// SYNTAX TEST "Step7 AWL.sublime-syntax"

// ==================================================
//  common
//  Performance: 3.0ms
// ==================================================

///////////////////////////////////////////////////////////////////////////////
// datatypes                                                                 //
///////////////////////////////////////////////////////////////////////////////

  TYPE "UDT_TypeName"
//^^^^^^^^^^^^^^^^^^^^ meta.block.udt.header
//^^^^ keyword.other.udt.begin
//     ^ punctuation.definition.string.begin
//     ^^^^^^^^^^^^^^ string.quoted.double
//                  ^ punctuation.definition.string.end
   { S7_language illegal := '7(1) Deutsch (Deutschland)  19.01.2014  10:33:55' }
// ^^^^^^^^^^^^^^^^^^^^^^^^^^^^^^^^^^^^^^^^^^^^^^^^^^^^^^^^^^^^^^^^^^^^^^^^^^^^^ meta.block.udt.header
// ^ meta.mapping - meta.mapping.key - meta.mapping.value
//  ^^^^^^^^^^^^^^^^^^^^^ meta.mapping.key - meta.mapping.value
//                       ^^ meta.mapping - meta.mapping.key - meta.mapping.value
//                         ^^^^^^^^^^^^^^^^^^^^^^^^^^^^^^^^^^^^^^^^^^^^^^^^^^^^ meta.mapping.value
//                                                                             ^ meta.mapping - meta.mapping.key - meta.mapping.value
// ^ punctuation.section.mapping.begin
//   ^^^^^^^^^^^ variable.annotation
//               ^^^^^^^ invalid.illegal.separator-expected
//                       ^^ punctuation.separator.key-value
//                                                                             ^ punctuation.section.mapping.end
   NON_RETAIN
// ^^^^^^^^^^ invalid.illegal
   READ_ONLY
// ^^^^^^^^^ invalid.illegal
   VERSION : 1.0
// ^^^^^^^^^^^^^ meta.block.udt.header
// ^^^^^^^^^ meta.mapping.key - meta.mapping.value
//          ^^^^ meta.mapping.value
// ^^^^^^^ entity.other.attribute-name
//         ^ punctuation.separator.key-value
//           ^ constant.numeric.float.version.major
//            ^ punctuation.separator.decimal.version
//             ^ constant.numeric.float.version.minor
   AUTHOR : name
// ^^^^^^^^^^^^^ meta.block.udt.header
// ^^^^^^^^ meta.mapping.key - meta.mapping.value
//         ^^^^^ meta.mapping.value
// ^^^^^^ entity.other.attribute-name
//        ^ punctuation.separator.key-value
//          ^^^^ string.unquoted
   FAMILY : name
// ^^^^^^^^^^^^^ meta.block.udt.header
// ^^^^^^^^ meta.mapping.key - meta.mapping.value
//         ^^^^^ meta.mapping.value
// ^^^^^^ entity.other.attribute-name
//        ^ punctuation.separator.key-value
//          ^^^^ string.unquoted
   NAME : name
// ^^^^^^^^^^^ meta.block.udt.header
// ^^^^^^ meta.mapping.key - meta.mapping.value
//       ^^^^^ meta.mapping.value
// ^^^^ entity.other.attribute-name
//      ^ punctuation.separator.key-value
//        ^^^^ string.unquoted
   ILLEGAL : unknown
// ^^^^^^^^^^^^^^^^^ meta.block.udt.header
// ^^^^^^^ invalid.illegal
//         ^ invalid.illegal
//           ^^^^^^^ invalid.illegal
  STRUCT
//^^^^^^^ meta.block.udt.header meta.struct
//^^^^^^ storage.type.struct.begin
     ID  : INT := 20 ;  //integer
// ^^^^^^^^^^^^^^^^^^^^^^^^^^^^^^^ meta.block.udt.header.s7.awl meta.struct.s7.awl
//   ^^^^^ meta.definition.variable - meta.definition.variable.storage
//        ^^^^^ meta.definition.variable.storage
//             ^^ meta.definition.variable - meta.definition.variable.storage - meta.definition.variable.value
//               ^^^^ meta.definition.variable.value
//   ^^ variable.other
//       ^ punctuation.separator.key-value
//         ^^^ storage.type.integer
//             ^^ keyword.operator.assignment
//                ^^ constant.numeric.integer
//                   ^ punctuation.terminator.statement
//                    ^^ - invalid
//                      ^^^^^^^^^ comment.line.double-slash
//                               ^ - invalid
     PTR : POINTER := P#0.0;
// ^^^^^^^^^^^^^^^^^^^^^^^^^^ meta.block.udt.header.s7.awl meta.struct.s7.awl
//   ^^^^^ meta.definition.variable.s7.awl
//        ^^^^^^^^^ meta.definition.variable.storage.s7.awl
//                 ^^ meta.definition.variable.s7.awl
//                   ^^^^^^ meta.definition.variable.value.s7.awl
//   ^^^ variable.other.s7.awl
//       ^ punctuation.separator.key-value.s7.awl
//         ^^^^^^^ storage.type.pointer.s7.awl
//                 ^^ keyword.operator.assignment.s7.awl
//                    ^^^^^ constant.language.pointer.s7.awl
     TMR : TIMER := T0;
// ^^^^^^^^^^^^^^^^^^^^^ meta.block.udt.header.s7.awl meta.struct.s7.awl
//   ^^^^^ meta.definition.variable.s7.awl
//        ^^^^^^^ meta.definition.variable.storage.s7.awl
//               ^^ meta.definition.variable.s7.awl
//                 ^^^ meta.definition.variable.value.s7.awl
//   ^^^ variable.other.s7.awl
//       ^ punctuation.separator.key-value.s7.awl
//         ^^^^^ storage.type.timer.s7.awl
//               ^^ keyword.operator.assignment.s7.awl
//                  ^^ variable.language.timer.s7.awl
  END_STRUCT ;
//^^^^^^^^^^^^^ meta.block.udt.header
//^^^^^^^^^^ meta.struct storage.type.struct.end
//           ^ punctuation.terminator.statement
  BEGIN
//^^^^^^ meta.block.udt.header
//^^^^^ invalid.illegal
  END_TYPE
//^^^^^^^^ meta.block.udt.header
//^^^^^^^^ keyword.other.udt.end

///////////////////////////////////////////////////////////////////////////////
// datablocks                                                                //
///////////////////////////////////////////////////////////////////////////////

  DATA_BLOCK "name" // comment
// ^^^^^^^^^^^^^^^^^^^^^^^^^^^ meta.block.db.header
// ^^^^^^^^^ keyword.other.db.begin
//           ^ punctuation.definition.string.begin
//           ^^^^^^ string.quoted.double
//            ^^^^ entity.name.block
//                  ^^ punctuation.definition.comment.begin
//                  ^^^^^^^^^^ comment.line.double-slash
   TITLE =the datablock description
// ^^^^^^^^^^^^^^^^^^^^^^^^^^^^^^^^ meta.block.db.header
// ^^^^^^^ meta.mapping.key - meta.mapping.value
//        ^^^^^^^^^^^^^^^^^^^^^^^^ meta.mapping.value - meta.mapping.key
// ^^^^^ entity.other.attribute-name.title
//       ^ punctuation.separator.key-value.title
//        ^^^^^^^^^^^^^^^^^^^^^^^^^ entity.name.section.s7.awl
   { S7_language illegal := '7(1) Deutsch (Deutschland)  19.01.2014  10:33:55' }
// ^^^^^^^^^^^^^^^^^^^^^^^^^^^^^^^^^^^^^^^^^^^^^^^^^^^^^^^^^^^^^^^^^^^^^^^^^^^^^ meta.block.db.header
// ^ meta.mapping - meta.mapping.key - meta.mapping.value
//  ^^^^^^^^^^^^^^^^^^^^^ meta.mapping.key - meta.mapping.value
//                       ^^ meta.mapping - meta.mapping.key - meta.mapping.value
//                         ^^^^^^^^^^^^^^^^^^^^^^^^^^^^^^^^^^^^^^^^^^^^^^^^^^^^ meta.mapping.value
//                                                                             ^ meta.mapping - meta.mapping.key - meta.mapping.value
// ^ punctuation.section.mapping.begin
//   ^^^^^^^^^^^ variable.annotation
//               ^^^^^^^ invalid.illegal.separator-expected
//                       ^^ punctuation.separator.key-value
//                                                                             ^ punctuation.section.mapping.end
   NON_RETAIN
// ^^^^^^^^^^ entity.other.attribute-name
   READ_ONLY
// ^^^^^^^^^ entity.other.attribute-name
   VERSION : 1.0
// ^^^^^^^^^^^^^ meta.block.db.header
// ^^^^^^^^^ meta.mapping.key - meta.mapping.value
//          ^^^^ meta.mapping.value
// ^^^^^^^ entity.other.attribute-name
//         ^ punctuation.separator.key-value
//           ^ constant.numeric.float.version.major
//            ^ punctuation.separator.decimal.version
//             ^ constant.numeric.float.version.minor
   AUTHOR : name
// ^^^^^^^^^^^^^ meta.block.db.header
// ^^^^^^^^ meta.mapping.key - meta.mapping.value
//         ^^^^^ meta.mapping.value
// ^^^^^^ entity.other.attribute-name
//        ^ punctuation.separator.key-value
//          ^^^^ string.unquoted
   FAMILY : name
// ^^^^^^^^^^^^^ meta.block.db.header
// ^^^^^^^^ meta.mapping.key - meta.mapping.value
//         ^^^^^ meta.mapping.value
// ^^^^^^ entity.other.attribute-name
//        ^ punctuation.separator.key-value
//          ^^^^ string.unquoted
   NAME : name
// ^^^^^^^^^^^ meta.block.db.header
// ^^^^^^ meta.mapping.key - meta.mapping.value
//       ^^^^^ meta.mapping.value
// ^^^^ entity.other.attribute-name
//      ^ punctuation.separator.key-value
//        ^^^^ string.unquoted
   ILLEGAL : unknown
// ^^^^^^^^^^^^^^^^^ meta.block.db.header
// ^^^^^^^ invalid.illegal
//         ^ invalid.illegal
//           ^^^^^^^ invalid.illegal

   "UDT_TypeName"
//<- meta.block.db.header
// ^^^^^^^^^^^^^^ meta.block.db.header
// ^ string.quoted.double punctuation.definition.string.begin
// ^^^^^^^^^^^^^^ meta.string
//  ^^^^^^^^^^^^ variable.other.symbol - string
//              ^ string.quoted.double punctuation.definition.string.end
   BEGIN illegal // comment
//<- meta.block.db.header
//^ meta.block.db.header - meta.block.db.body
// ^^^^^^^^^^^^^^^^^^^^^^^^ meta.block.db.body - meta.block.db.header
// ^^^^^ keyword.other.begin
//       ^^^^^^^ invalid.illegal
//               ^^ punctuation.definition.comment.begin
//               ^^^^^^^^^^ comment.line.double-slash

   VAR[0].child[ 0 ].attr := W#16#0 ;  // comment
//<- meta.block.db.body
//^^^^^^^^^^^^^^^^^^^^^^^^^^^^^^^^^^^^^^^^^^^^^^^ meta.block.db.body
//    ^^^ meta.brackets
//             ^^^^^ meta.brackets
// ^^^ variable.other.local
//    ^ punctuation.section.brackets.begin
//     ^ constant.numeric.integer
//      ^ punctuation.section.brackets.end
//       ^ punctuation.accessor.dot
//        ^^^^^ variable.other.member
//             ^ punctuation.section.brackets.begin
//               ^ constant.numeric.integer
//                 ^ punctuation.section.brackets.end
//                  ^ punctuation.accessor.dot
//                   ^^^^ variable.other.member
//                        ^^ keyword.operator.assignment
//                           ^^^^^^ constant.numeric.integer.hexadecimal
//                                  ^ punctuation.terminator.statement
   test := W#16 ; illegal // comment
// ^^^^ variable.other.local
//      ^^ keyword.operator.assignment
//         ^^^^ invalid.illegal
//             ^ - invalid
//              ^ punctuation.terminator.statement
//               ^ - invalid
//                ^^^^^^^^ invalid.illegal.eol-expected
//                        ^^ punctuation.definition.comment.begin
//                        ^^^^^^^^^^ comment.line.double-slash
   incomplete
   next_is_valid
// ^^^^^^^^^^^^^ variable.other.local
   date_time := DT#90-1-1-0:0:0.000;
//              ^^^^^^^^^^^^^^^^^^^ constant.language.datetime
//              ^^^ storage.type.numeric.s7.awl
//                   ^ punctuation.separator.date
//                     ^ punctuation.separator.date
//                       ^ punctuation.separator.date
//                         ^ punctuation.separator.time
//                           ^ punctuation.separator.time
//                             ^ punctuation.separator.time
   date_time := DT#2017-12-31-23:59:59.999;
//              ^^^^^^^^^^^^^^^^^^^^^^^^^^ constant.language.datetime
//              ^^^ storage.type.numeric.s7.awl
//                     ^ punctuation.separator.date
//                        ^ punctuation.separator.date
//                           ^ punctuation.separator.date
//                              ^ punctuation.separator.time
//                                 ^ punctuation.separator.time
//                                    ^ punctuation.separator.time
   date_time := DT#2017;
//              ^^^^^^^ invalid.illegal
   END_DATA_BLOCK
//<- meta.block.db.body
//^^^^^^^^^^^^^^^ meta.block.db.body
// ^^^^^^^^^^^^^^ keyword.other.db.end

///////////////////////////////////////////////////////////////////////////////
// functions                                                                 //
///////////////////////////////////////////////////////////////////////////////

   FUNCTION "name" : INT  // comment
// ^^^^^^^^^^^^^^^^^^^^^^^^^^^^^^^^^^ meta.block.fc.header
// ^^^^^^^^ keyword.other.fc.begin
//          ^ punctuation.definition.string.begin
//          ^^^^^^ string.quoted.double
//           ^^^^ entity.name.block
//                 ^ punctuation.separator.mapping.pair
//                   ^^^ storage.type.integer
//                        ^^ punctuation.definition.comment.begin
//                        ^^^^^^^^^^ comment.line.double-slash
   TITLE =the function description
// ^^^^^^^^^^^^^^^^^^^^^^^^^^^^^^^ meta.block.fc.header
// ^^^^^^^ meta.mapping.key - meta.mapping.value
//        ^^^^^^^^^^^^^^^^^^^^^^^^ meta.mapping.value - meta.mapping.key
// ^^^^^ entity.other.attribute-name.title
//       ^ punctuation.separator.key-value.title
//        ^^^^^^^^^^^^^^^^^^^^^^^^ entity.name.section.s7.awl
   { S7_language illegal := '7(1) Deutsch (Deutschland)  19.01.2014  10:33:55' }
// ^^^^^^^^^^^^^^^^^^^^^^^^^^^^^^^^^^^^^^^^^^^^^^^^^^^^^^^^^^^^^^^^^^^^^^^^^^^^^ meta.block.fc.header
// ^ meta.mapping - meta.mapping.key - meta.mapping.value
//  ^^^^^^^^^^^^^^^^^^^^^ meta.mapping.key - meta.mapping.value
//                       ^^ meta.mapping - meta.mapping.key - meta.mapping.value
//                         ^^^^^^^^^^^^^^^^^^^^^^^^^^^^^^^^^^^^^^^^^^^^^^^^^^^^ meta.mapping.value
//                                                                             ^ meta.mapping - meta.mapping.key - meta.mapping.value
// ^ punctuation.section.mapping.begin
//   ^^^^^^^^^^^ variable.annotation
//               ^^^^^^^ invalid.illegal.separator-expected
//                       ^^ punctuation.separator.key-value
//                                                                             ^ punctuation.section.mapping.end
   VERSION : 1.0
// ^^^^^^^^^^^^^ meta.block.fc.header
// ^^^^^^^^^ meta.mapping.key - meta.mapping.value
//          ^^^^ meta.mapping.value
// ^^^^^^^ entity.other.attribute-name
//         ^ punctuation.separator.key-value
//           ^ constant.numeric.float.version.major
//            ^ punctuation.separator.decimal.version
//             ^ constant.numeric.float.version.minor
   AUTHOR : name
// ^^^^^^^^^^^^^ meta.block.fc.header
// ^^^^^^^^ meta.mapping.key - meta.mapping.value
//         ^^^^^ meta.mapping.value
// ^^^^^^ entity.other.attribute-name
//        ^ punctuation.separator.key-value
//          ^^^^ string.unquoted
   FAMILY : name
// ^^^^^^^^^^^^^ meta.block.fc.header
// ^^^^^^^^ meta.mapping.key - meta.mapping.value
//         ^^^^^ meta.mapping.value
// ^^^^^^ entity.other.attribute-name
//        ^ punctuation.separator.key-value
//          ^^^^ string.unquoted
   NAME : name
// ^^^^^^^^^^^ meta.block.fc.header
// ^^^^^^ meta.mapping.key - meta.mapping.value
//       ^^^^^ meta.mapping.value
// ^^^^ entity.other.attribute-name
//      ^ punctuation.separator.key-value
//        ^^^^ string.unquoted
   ILLEGAL : unknown
// ^^^^^^^^^^^^^^^^^ meta.block.fc.header
// ^^^^^^^ invalid.illegal
//         ^ invalid.illegal
//           ^^^^^^^ invalid.illegal

   VAR_INPUT illegal // comment
// <- meta.block.fc.header - meta.block.fc.body
// ^^^^^^^^^^^^^^^^^^^^^^^^^^^^^ meta.block.fc.header meta.block.var.input
// ^^^^^^^^^ keyword.control.var.input.begin
//           ^^^^^^^ invalid.illegal.eol-expected
//                   ^^^^^^^^^^ comment.line.double-slash
     RUN : BOOL := TRUE ;  //bool
// ^^^^^^^^^^^^^^^^^^^^^^^^^^^^^^^ meta.block.fc.header meta.block.var.input
//   ^^^^^ meta.definition.variable - meta.definition.variable.storage
//        ^^^^^^ meta.definition.variable.storage - meta.definition.variable.value
//              ^^ meta.definition.variable - meta.definition.variable.storage - meta.definition.variable.value
//                ^^^^^^ meta.definition.variable.value - meta.definition.variable.storage
//   ^^^ variable.other
//       ^ punctuation.separator.key-value
//         ^^^^ storage.type.bool
//              ^^ keyword.operator.assignment
//                 ^^^^ constant.language.boolean
//                      ^ punctuation.terminator.statement
//                       ^^ - invalid
//                         ^^^^^^ comment.line.double-slash
//                               ^ - invalid
     ID  : INT  ;  //integer
// ^^^^^^^^^^^^^^^^^^^^^^^^^ meta.block.fc.header meta.block.var.input
//   ^^^^^ meta.definition.variable - meta.definition.variable.storage
//        ^^^^^^ meta.definition.variable.storage
//   ^^ variable.other
//       ^ punctuation.separator.key-value
//         ^^^ storage.type.integer
//              ^ punctuation.terminator.statement
//               ^^ - invalid
//                 ^^^^^^^^^ comment.line.double-slash
//                          ^ - invalid
     _S1  : STRING[32] ;  //string
// ^^^^^^^^^^^^^^^^^^^^^^^^^^^^^^^ meta.block.fc.header meta.block.var.input
//   ^^^^^ meta.definition.variable - meta.definition.variable.storage
//         ^^^^^^^^^^^^ meta.definition.variable.storage
//   ^^^ variable.other
//        ^ punctuation.separator.key-value
//          ^^^^^^^^^^ storage.type.string
//                     ^ punctuation.terminator.statement
//                      ^^ - invalid
//                        ^^^^^^^^ comment.line.double-slash
//                                ^ - invalid
     _AR  : ARRAY[ 0 .. 20 ] OF //array
// ^^^^^^^^^^^^^^^^^^^^^^^^^^^^^^^^^^^^ meta.block.fc.header meta.block.var.input
//   ^^^^^ meta.definition.variable - meta.definition.variable.storage
//         ^^^^^^^^^^^^^^^^^^^^^^^^^^^^ meta.definition.variable.storage
//          ^^^^^^^^^^^^^^^^^^^^^^^^^^^ meta.sequence.array
//   ^^^ variable.other
//        ^ punctuation.separator.key-value
//          ^^^^^ storage.type.array
//               ^ punctuation.definition.array.begin
//                 ^ constant.numeric.integer
//                   ^^ keyword.operator.range
//                      ^^ constant.numeric.integer
//                         ^ punctuation.definition.array.end
//                          ^ - invalid
//                           ^^ keyword.control.of
//                             ^ - invalid
//                              ^^ punctuation.definition.comment.begin
//                              ^^^^^^^ comment.line.double-slash
//                                     ^ - invalid
            DWORD := [ DW#16#0, DW#16#2, DW#16#A ] ;  //integer
//^^^^^^^^^^^^^^^^^^^^^^^^^^^^^^^^^^^^^^^^^^^^^^^^^^^^^^^^^^^^^^ meta.block.fc.header meta.block.var.input
//^^^^^^^^^^^^^^^^ meta.definition.variable.storage
//^^^^^^^^^^^^^^^ meta.sequence.array
//               ^^^^ - meta.sequence
//                   ^^^^^^^^^^^^^^^^^^^^^^^^^^^^^ meta.sequence.list.s7.awl
//                                                ^ - meta.sequence
//          ^^^^^ storage.type.dword
//                ^^ keyword.operator.assignment
//                   ^ punctuation.section.sequence.begin
//                     ^^^^^^^ constant.numeric.integer.hexadecimal
//                            ^ punctuation.separator.sequence
//                              ^^^^^^^ constant.numeric.integer.hexadecimal
//                                     ^ punctuation.separator.sequence
//                                       ^^^^^^^ constant.numeric.integer.hexadecimal
//                                               ^ punctuation.section.sequence.end
//                                                ^ - invalid
//                                                 ^ punctuation.terminator.statement
//                                                  ^^ - invalid
//                                                    ^^^^^^^^^ comment.line.double-slash
//                                                             ^ - invalid
     _ST  : STRUCT  //structure
// ^^^^^^^^^^^^^^^^^^^^^^^^^^^^ meta.block.fc.header meta.block.var.input
//   ^^^^^ meta.definition.variable - meta.definition.variable.storage
//         ^^^^^^^^^^^^^^^^^^^^ meta.definition.variable.storage
//          ^^^^^^^^^^^^^^^^^^^ meta.struct
//   ^^^ variable.other
//        ^ punctuation.separator.key-value
//          ^^^^^^ storage.type.struct.begin
//                  ^^ comment.line.double-slash
//                  ^^^^^^^^^^^ comment.line.double-slash
//                             ^ - invalid
       RUN : BOOL ;  //bool
// ^^^^^^^^^^^^^^^^^^^^^^^^ meta.block.fc.header meta.block.var.input meta.definition.variable.storage meta.struct
//     ^^^^^ meta.definition.variable
//          ^^^^^^ meta.definition.variable.storage meta.definition.variable.storage
//     ^^^ variable.other
//         ^ punctuation.separator.key-value
//           ^^^^ storage.type.bool
//                ^ punctuation.terminator.statement
//                 ^^ - invalid
//                   ^^^^^^ comment.line.double-slash
//                         ^ - invalid
       ID  : INT  ;  //integer
// ^^^^^^^^^^^^^^^^^^^^^^^^^^^ meta.block.fc.header meta.block.var.input meta.definition.variable.storage meta.struct
//     ^^^^^ meta.definition.variable
//          ^^^^^^ meta.definition.variable.storage meta.definition.variable.storage
//     ^^ variable.other
//         ^ punctuation.separator.key-value
//           ^^^ storage.type.integer
//                ^ punctuation.terminator.statement
//                 ^^ - invalid
//                   ^^^^^^^^^ comment.line.double-slash
//                            ^ - invalid
       _S1  : STRING[32] := 'initial';  //string
// ^^^^^^^^^^^^^^^^^^^^^^^^^^^^^^^^^^^^^^^^^^^^^^ meta.block.fc.header meta.block.var.input meta.definition.variable.storage meta.struct
//     ^^^^^^ meta.definition.variable
//           ^^^^^^^^^^^^ meta.definition.variable.storage meta.definition.variable.storage
//                       ^^ meta.definition.variable.storage meta.definition.variable
//                         ^^^^^^^^^^ meta.definition.variable.storage meta.definition.variable.value
//     ^^^ variable.other
//          ^ punctuation.separator.key-value
//            ^^^^^^^^^^ storage.type.string
//                       ^^ keyword.operator.assignment.s7.awl
//                          ^^^^^^^^^ string.quoted.single.s7.awl
//                                   ^ punctuation.terminator.statement
//                                    ^^ - invalid
//                                      ^^^^^^^^ comment.line.double-slash
//                                              ^ - invalid
       _V   : FLOAT := -1.2 ;
// ^^^^^^^^^^^^^^^^^^^^^^^^^^ meta.block.fc.header meta.block.var.input meta.definition.variable.storage meta.struct
//     ^^^^^^ meta.definition.variable
//           ^^^^^^^ meta.definition.variable.storage meta.definition.variable.storage
//                  ^^ meta.definition.variable.storage meta.definition.variable
//                    ^^^^^^ meta.definition.variable.storage meta.definition.variable.value
//     ^^ variable.other
//          ^ punctuation.separator.key-value
//            ^^^^^ storage.type.other.s7.awl
//                  ^^ keyword.operator.assignment.s7.awl
//                     ^^^^ constant.numeric.float.decimal.s7.awl
//                          ^ punctuation.terminator.statement
//                           ^^ - invalid
    END_STRUCT ;
// ^^^^^^^^^^^^^ meta.block.fc.header meta.block.var.input
// ^^^^^^^^^^^^ meta.definition.variable.storage
// ^^^^^^^^^^^ meta.struct
//  ^^^^^^^^^^ storage.type.struct.end
//             ^ punctuation.terminator.statement
     _AS  : ARRAY[0..20] OF STRUCT //array
// ^^^^^^^^^^^^^^^^^^^^^^^^^^^^^^^^^^^^^^^^ meta.block.fc.header meta.block.var.input
//   ^^^^^ meta.definition.variable - meta.definition.variable.storage
//         ^^^^^^^^^^^^^^^^^^^^^^^^^^^^^^^ meta.definition.variable.storage
//          ^^^^^^^^^^^^^^^^^^^^^^^^^^^^^^ meta.sequence.array
//                          ^^^^^^^^^^^^^^ meta.struct
//   ^^^ variable.other
//        ^ punctuation.separator.key-value
//          ^^^^^ storage.type.array
//               ^ punctuation.definition.array.begin
//                ^ constant.numeric.integer
//                 ^^ keyword.operator.range
//                   ^^ constant.numeric.integer
//                     ^ punctuation.definition.array.end
//                       ^^ keyword.control.of
//                          ^^^^^^ storage.type.struct.begin
//                                 ^^ punctuation.definition.comment.begin
//                                 ^^^^^^^ comment.line.double-slash
       RUN : BOOL ;  //bool
// ^^^^^^^^^^^^^^^^^^^^^^^^ meta.block.fc.header meta.block.var.input meta.definition.variable.storage meta.sequence.array meta.struct
//     ^^^^^ meta.definition.variable
//          ^^^^^^ meta.definition.variable.storage meta.definition.variable.storage
//     ^^^ variable.other
//         ^ punctuation.separator.key-value
//           ^^^^ storage.type.bool
//                ^ punctuation.terminator.statement
//                 ^^ - invalid
//                   ^^^^^^ comment.line.double-slash
//                         ^ - invalid
       ID  : INT  ;  //integer
// ^^^^^^^^^^^^^^^^^^^^^^^^^^^ meta.block.fc.header meta.block.var.input meta.definition.variable.storage meta.sequence.array meta.struct
//     ^^^^^ meta.definition.variable
//          ^^^^^^ meta.definition.variable.storage meta.definition.variable.storage
//     ^^ variable.other
//         ^ punctuation.separator.key-value
//           ^^^ storage.type.integer
//                ^ punctuation.terminator.statement
//                 ^^ - invalid
//                   ^^^^^^^^^ comment.line.double-slash
//                            ^ - invalid
       _S1  : STRING[32] ;  //string
// ^^^^^^^^^^^^^^^^^^^^^^^^^^^^^^^^^ meta.block.fc.header meta.block.var.input meta.definition.variable.storage meta.sequence.array meta.struct
//     ^^^^^ meta.definition.variable
//           ^^^^^^^^^^^ meta.definition.variable.storage meta.definition.variable.storage
//     ^^^ variable.other
//          ^ punctuation.separator.key-value
//            ^^^^^^^^^^ storage.type.string
//                       ^ punctuation.terminator.statement
//                        ^^ - invalid
//                          ^^^^^^^^ comment.line.double-slash
//                                  ^ - invalid
    END_STRUCT ;
//^^^^^^^^^^^^^^ meta.block.fc.header meta.block.var.input
//^^^^^^^^^^^^^ meta.definition.variable.storage
//^^^^^^^^^^^^ meta.struct
//  ^^^^^^^^^^ storage.type.struct.end
//             ^ punctuation.terminator.statement
   END_VAR
// <- meta.block.fc.header meta.block.var.input
// ^^^^^^^ meta.block.fc.header meta.block.var.input
// ^^^^^^^ keyword.control.var.end

   VAR_OUTPUT
// <- meta.block.fc.header - meta.block.fc.body
// ^^^^^^^^^^ meta.block.fc.header meta.block.var.output
// ^^^^^^^^^^ keyword.control.var.output.begin
     RUN : BOOL ;  //bool
// ^^^^^^^^^^^^^^^^^^^^^^ meta.block.fc.header meta.block.var.output
//   ^^^^^ meta.definition.variable - meta.definition.variable.storage
//        ^^^^^^ meta.definition.variable.storage
//   ^^^ variable.other
//       ^ punctuation.separator.key-value
//         ^^^^ storage.type.bool
//              ^ punctuation.terminator.statement
//               ^^ - invalid
//                 ^^^^^^ comment.line.double-slash
//                       ^ - invalid
     ID  : INT  ;  //integer
// ^^^^^^^^^^^^^^^^^^^^^^^^^ meta.block.fc.header meta.block.var.output
//   ^^^^^ meta.definition.variable - meta.definition.variable.storage
//        ^^^^^^ meta.definition.variable.storage
//   ^^ variable.other
//       ^ punctuation.separator.key-value
//         ^^^ storage.type.integer
//              ^ punctuation.terminator.statement
//               ^^ - invalid
//                 ^^^^^^^^^ comment.line.double-slash
//                          ^ - invalid
     _S1  : STRING[32] ;  //string
// ^^^^^^^^^^^^^^^^^^^^^^^^^^^^^^^ meta.block.fc.header meta.block.var.output
//   ^^^^^ meta.definition.variable - meta.definition.variable.storage
//         ^^^^^^^^^^^^ meta.definition.variable.storage
//   ^^^ variable.other
//        ^ punctuation.separator.key-value
//          ^^^^^^^^^^ storage.type.string
//                     ^ punctuation.terminator.statement
//                      ^^ - invalid
//                        ^^^^^^^^ comment.line.double-slash
//                                ^ - invalid
     _AR  : ARRAY[ 0 .. 20 ] OF //array
// ^^^^^^^^^^^^^^^^^^^^^^^^^^^^^^^^^^^^ meta.block.fc.header meta.block.var.output
//   ^^^^^ meta.definition.variable - meta.definition.variable.storage
//         ^^^^^^^^^^^^^^^^^^^^^^^^^^^^ meta.definition.variable.storage
//          ^^^^^^^^^^^^^^^^^^^^^^^^^^^ meta.sequence.array
//   ^^^ variable.other
//        ^ punctuation.separator.key-value
//          ^^^^^ storage.type.array
//               ^ punctuation.definition.array.begin
//                 ^ constant.numeric.integer
//                   ^^ keyword.operator.range
//                      ^^ constant.numeric.integer
//                         ^ punctuation.definition.array.end
//                           ^^ keyword.control.of
//                              ^^ punctuation.definition.comment.begin
//                              ^^^^^^^ comment.line.double-slash
            DWORD ;  //integer
// ^^^^^^^^^^^^^^^^^^^^^^^^^^^ meta.block.fc.header meta.block.var.output
// ^^^^^^^^^^^^^^ meta.definition.variable.storage meta.sequence.array
//          ^^^^^ storage.type.dword
//                   ^^^^^^^^^ comment.line.double-slash
//                            ^ - invalid
     _ST  : STRUCT  //structure
// ^^^^^^^^^^^^^^^^^^^^^^^^^^^^ meta.block.fc.header meta.block.var.output
//   ^^^^^ meta.definition.variable - meta.definition.variable.storage
//         ^^^^^^^^^^^^^^^^^^^^ meta.definition.variable.storage
//          ^^^^^^^^^^^^^^^^^^^ meta.struct
//   ^^^ variable.other
//        ^ punctuation.separator.key-value
//          ^^^^^^ storage.type.struct.begin
//                  ^^^^^^^^^^^ comment.line.double-slash
//                             ^ - invalid
       RUN : BOOL ;  //bool
// ^^^^^^^^^^^^^^^^^^^^^^^^ meta.block.fc.header meta.block.var.output meta.definition.variable.storage meta.struct
//     ^^^^^ meta.definition.variable
//          ^^^^^^ meta.definition.variable.storage meta.definition.variable.storage
//     ^^^ variable.other
//         ^ punctuation.separator.key-value
//           ^^^^ storage.type.bool
//                ^ punctuation.terminator.statement
//                   ^^^^^^ comment.line.double-slash
//                         ^ - invalid
       ID  : INT  ;  //integer
// ^^^^^^^^^^^^^^^^^^^^^^^^^^^ meta.block.fc.header meta.block.var.output meta.definition.variable.storage meta.struct
//     ^^^^^ meta.definition.variable
//          ^^^^^^ meta.definition.variable.storage meta.definition.variable.storage
//     ^^ variable.other
//         ^ punctuation.separator.key-value
//           ^^^ storage.type.integer
       _S1  : STRING[32] ;  //string
// ^^^^^^^^^^^^^^^^^^^^^^^^^^^^^^^^^ meta.block.fc.header meta.block.var.output meta.definition.variable.storage meta.struct
//     ^^^^^ meta.definition.variable
//           ^^^^^^^^^^^ meta.definition.variable.storage meta.definition.variable.storage
//     ^^^ variable.other
//          ^ punctuation.separator.key-value
//            ^^^^^^^^^^ storage.type.string
    END_STRUCT ;
//^^^^^^^^^^^^^^^ meta.block.fc.header meta.block.var.output
//^^^^^^^^^^^^^ meta.definition.variable.storage
//^^^^^^^^^^^^ meta.struct
//  ^^^^^^^^^^ storage.type.struct.end
//             ^ punctuation.terminator.statement
//              ^ - invalid
     _AS  : ARRAY[ 0 .. 20 ] OF STRUCT //array
// ^^^^^^^^^^^^^^^^^^^^^^^^^^^^^^^^^^^^^^^^^^^ meta.block.fc.header meta.block.var.output
//   ^^^^^ meta.definition.variable - meta.definition.variable.storage
//         ^^^^^^^^^^^^^^^^^^^^^^^^^^^^^^^^^^^ meta.definition.variable.storage
//          ^^^^^^^^^^^^^^^^^^^^^^^^^^^^^^^^^^ meta.sequence.array
//                              ^^^^^^^^^^^^^^ meta.struct
//   ^^^ variable.other
//        ^ punctuation.separator.key-value
//          ^^^^^ storage.type.array
//               ^ punctuation.definition.array.begin
//                 ^ constant.numeric.integer
//                   ^^ keyword.operator.range
//                      ^^ constant.numeric.integer
//                         ^ punctuation.definition.array.end
//                           ^^ keyword.control.of
//                              ^^^^^^ storage.type.struct.begin
//                                     ^^ punctuation.definition.comment.begin
//                                     ^^^^^^^ comment.line.double-slash
//                                            ^ - invalid
       RUN : BOOL ;  //bool
// ^^^^^^^^^^^^^^^^^^^^^^^^ meta.block.fc.header meta.block.var.output meta.definition.variable.storage meta.sequence.array meta.struct
//     ^^^^^ meta.definition.variable
//          ^^^^^^ meta.definition.variable.storage meta.definition.variable.storage
//     ^^^ variable.other
//         ^ punctuation.separator.key-value
//           ^^^^ storage.type.bool
       ID  : INT  ;  //integer
// ^^^^^^^^^^^^^^^^^^^^^^^^^^^ meta.block.fc.header meta.block.var.output meta.definition.variable.storage meta.sequence.array meta.struct
//     ^^^^^ meta.definition.variable
//          ^^^^^^ meta.definition.variable.storage meta.definition.variable.storage
//     ^^ variable.other
//         ^ punctuation.separator.key-value
//           ^^^ storage.type.integer
       _S1  : STRING[32] ;  //string
// ^^^^^^^^^^^^^^^^^^^^^^^^^^^^^^^^^ meta.block.fc.header meta.block.var.output meta.definition.variable.storage meta.sequence.array meta.struct
//     ^^^^^ meta.definition.variable
//           ^^^^^^^^^^^ meta.definition.variable.storage meta.definition.variable.storage
//     ^^^ variable.other
//          ^ punctuation.separator.key-value
//            ^^^^^^^^^^ storage.type.string
    END_STRUCT ;
//^^^^^^^^^^^^^^^ meta.block.fc.header meta.block.var
//^^^^^^^^^^^^^ meta.definition.variable.storage
//^^^^^^^^^^^^ meta.struct
//  ^^^^^^^^^^ storage.type.struct.end
//             ^ punctuation.terminator.statement
//              ^ - invalid
   END_VAR
// <- meta.block.fc.header meta.block.var.output
// ^^^^^^^ meta.block.fc.header meta.block.var.output
// ^^^^^^^ keyword.control.var.end

   VAR_IN_OUT
// <- meta.block.fc.header - meta.block.fc.body
// ^^^^^^^^^^ meta.block.fc.header meta.block.var.in-out
// ^^^^^^^^^^ keyword.control.var.in-out.begin
     RUN : BOOL ;  //bool
// ^^^^^^^^^^^^^^^^^^^^^^ meta.block.fc.header meta.block.var.in-out
//   ^^^^^ meta.definition.variable - meta.definition.variable.storage
//        ^^^^^^ meta.definition.variable.storage
//   ^^^ variable.other
//       ^ punctuation.separator.key-value
//         ^^^^ storage.type.bool
     ID  : INT  ;  //integer
// ^^^^^^^^^^^^^^^^^^^^^^^^^ meta.block.fc.header meta.block.var.in-out
//   ^^^^^ meta.definition.variable - meta.definition.variable.storage
//        ^^^^^^ meta.definition.variable.storage
//   ^^ variable.other
//       ^ punctuation.separator.key-value
//         ^^^ storage.type.integer
     _S1  : STRING[32] ;  //string
// ^^^^^^^^^^^^^^^^^^^^^^^^^^^^^^^ meta.block.fc.header meta.block.var.in-out
//   ^^^^^ meta.definition.variable - meta.definition.variable.storage
//         ^^^^^^^^^^^^ meta.definition.variable.storage
//   ^^^ variable.other
//        ^ punctuation.separator.key-value
//          ^^^^^^^^^^ storage.type.string
     _AR  : ARRAY[ 0 .. 20 ] OF //array
// ^^^^^^^^^^^^^^^^^^^^^^^^^^^^^^^^^^^^ meta.block.fc.header meta.block.var.in-out
//   ^^^^^ meta.definition.variable - meta.definition.variable.storage
//         ^^^^^^^^^^^^^^^^^^^^^^^^^^^^ meta.definition.variable.storage
//          ^^^^^^^^^^^^^^^^^^^^^^^^^^^ meta.sequence.array
//   ^^^ variable.other
//        ^ punctuation.separator.key-value
//          ^^^^^ storage.type.array
//               ^ punctuation.definition.array.begin
//                 ^ constant.numeric.integer
//                   ^^ keyword.operator.range
//                      ^^ constant.numeric.integer
//                         ^ punctuation.definition.array.end
//                           ^^ keyword.control.of
//                              ^^ punctuation.definition.comment.begin
//                              ^^^^^^^ comment.line.double-slash
            DWORD ;  //integer
// ^^^^^^^^^^^^^^^^^^^^^^^^^^^ meta.block.fc.header meta.block.var.in-out
// ^^^^^^^^^^^^^^ meta.definition.variable.storage meta.sequence.array
//          ^^^^^ storage.type.dword
     _ST  : STRUCT  //structure
// ^^^^^^^^^^^^^^^^^^^^^^^^^^^^ meta.block.fc.header meta.block.var.in-out
//   ^^^^^ meta.definition.variable - meta.definition.variable.storage
//         ^^^^^^^^^^^^^^^^^^^^ meta.definition.variable.storage
//          ^^^^^^^^^^^^^^^^^^^ meta.struct
//   ^^^ variable.other
//        ^ punctuation.separator.key-value
//          ^^^^^^ storage.type.struct.begin
       RUN : BOOL ;  //bool
// ^^^^^^^^^^^^^^^^^^^^^^^^ meta.block.fc.header meta.block.var.in-out meta.definition.variable.storage meta.struct
//     ^^^^^ meta.definition.variable
//          ^^^^^^ meta.definition.variable.storage meta.definition.variable.storage
//     ^^^ variable.other
//         ^ punctuation.separator.key-value
//           ^^^^ storage.type.bool
       ID  : INT  ;  //integer
// ^^^^^^^^^^^^^^^^^^^^^^^^^^^ meta.block.fc.header meta.block.var.in-out meta.definition.variable.storage meta.struct
//     ^^^^^ meta.definition.variable
//          ^^^^^^ meta.definition.variable.storage meta.definition.variable.storage
//     ^^ variable.other
//         ^ punctuation.separator.key-value
//           ^^^ storage.type.integer
       _S1  : STRING[32] ;  //string
// ^^^^^^^^^^^^^^^^^^^^^^^^^^^^^^^^^ meta.block.fc.header meta.block.var.in-out meta.definition.variable.storage meta.struct
//     ^^^^^ meta.definition.variable
//           ^^^^^^^^^^^ meta.definition.variable.storage meta.definition.variable.storage
//     ^^^ variable.other
//          ^ punctuation.separator.key-value
//            ^^^^^^^^^^ storage.type.string
    END_STRUCT ;
//^^^^^^^^^^^^^^^ meta.block.fc.header meta.block.var.in-out
//^^^^^^^^^^^^^ meta.definition.variable.storage
//^^^^^^^^^^^^ meta.struct
//  ^^^^^^^^^^ storage.type.struct.end
//             ^ punctuation.terminator.statement
//              ^ - invalid
     _AS  : ARRAY[ 0 .. 20 ] OF STRUCT //array
// ^^^^^^^^^^^^^^^^^^^^^^^^^^^^^^^^^^^^^^^^^^^ meta.block.fc.header meta.block.var.in-out
//   ^^^^^ meta.definition.variable - meta.definition.variable.storage
//         ^^^^^^^^^^^^^^^^^^^^^^^^^^^^^^^^^^^ meta.definition.variable.storage
//          ^^^^^^^^^^^^^^^^^^^^^^^^^^^^^^^^^^ meta.sequence.array
//                              ^^^^^^^^^^^^^^ meta.struct
//   ^^^ variable.other
//        ^ punctuation.separator.key-value
//          ^^^^^ storage.type.array
//               ^ punctuation.definition.array.begin
//                 ^ constant.numeric.integer
//                   ^^ keyword.operator.range
//                      ^^ constant.numeric.integer
//                         ^ punctuation.definition.array.end
//                           ^^ keyword.control.of
//                              ^^^^^^ storage.type.struct.begin
//                                     ^^ punctuation.definition.comment.begin
//                                     ^^^^^^^ comment.line.double-slash
       RUN : BOOL ;  //bool
// ^^^^^^^^^^^^^^^^^^^^^^^^ meta.block.fc.header meta.block.var.in-out meta.definition.variable.storage meta.sequence.array meta.struct
//     ^^^^^ meta.definition.variable
//          ^^^^^^ meta.definition.variable.storage meta.definition.variable.storage
//     ^^^ variable.other
//         ^ punctuation.separator.key-value
//           ^^^^ storage.type.bool
       ID  : INT  ;  //integer
// ^^^^^^^^^^^^^^^^^^^^^^^^^^^ meta.block.fc.header meta.block.var.in-out meta.definition.variable.storage meta.sequence.array meta.struct
//     ^^^^^ meta.definition.variable
//          ^^^^^^ meta.definition.variable.storage meta.definition.variable.storage
//     ^^ variable.other
//         ^ punctuation.separator.key-value
//           ^^^ storage.type.integer
       _S1  : STRING[32] ;  //string
// ^^^^^^^^^^^^^^^^^^^^^^^^^^^^^^^^^ meta.block.fc.header meta.block.var.in-out meta.definition.variable.storage meta.sequence.array meta.struct
//     ^^^^^ meta.definition.variable
//           ^^^^^^^^^^^^ meta.definition.variable.storage meta.definition.variable.storage
//     ^^^ variable.other
//          ^ punctuation.separator.key-value
//            ^^^^^^^^^^ storage.type.string
    END_STRUCT ;
//^^^^^^^^^^^^^^^ meta.block.fc.header meta.block.var.in-out
//^^^^^^^^^^^^^ meta.definition.variable.storage
//^^^^^^^^^^^^ meta.struct
//  ^^^^^^^^^^ storage.type.struct.end
//             ^ punctuation.terminator.statement
   END_VAR
// <- meta.block.fc.header meta.block.var.in-out
// ^^^^^^^ meta.block.fc.header meta.block.var.in-out
// ^^^^^^^ keyword.control.var.end

   VAR_TEMP
// <- meta.block.fc.header - meta.block.fc.body
// ^^^^^^^^ meta.block.fc.header meta.block.var.temp
// ^^^^^^^^ keyword.control.var.temp.begin
     RUN : BOOL ;  //bool
// ^^^^^^^^^^^^^^^^^^^^^^ meta.block.fc.header meta.block.var.temp
//   ^^^^^ meta.definition.variable - meta.definition.variable.storage
//        ^^^^^^ meta.definition.variable.storage
//   ^^^ variable.other
//       ^ punctuation.separator.key-value
//         ^^^^ storage.type.bool
     ID  : INT  ;  //integer
// ^^^^^^^^^^^^^^^^^^^^^^^^^ meta.block.fc.header meta.block.var.temp
//   ^^^^^ meta.definition.variable - meta.definition.variable.storage
//        ^^^^^^ meta.definition.variable.storage
//   ^^ variable.other
//       ^ punctuation.separator.key-value
//         ^^^ storage.type.integer
     _S1  : STRING[32] ;  //string
// ^^^^^^^^^^^^^^^^^^^^^^^^^^^^^^^ meta.block.fc.header meta.block.var.temp
//   ^^^^^ meta.definition.variable - meta.definition.variable.storage
//         ^^^^^^^^^^^^ meta.definition.variable.storage
//   ^^^ variable.other
//        ^ punctuation.separator.key-value
//          ^^^^^^^^^^ storage.type.string
     _AR  : ARRAY[ 0 .. 20 ] OF //array
// ^^^^^^^^^^^^^^^^^^^^^^^^^^^^^^^^^^^^ meta.block.fc.header meta.block.var.temp
//   ^^^^^ meta.definition.variable - meta.definition.variable.storage
//         ^^^^^^^^^^^^^^^^^^^^^^^^^^^^ meta.definition.variable.storage
//          ^^^^^^^^^^^^^^^^^^^^^^^^^^^ meta.sequence.array
//   ^^^ variable.other
//        ^ punctuation.separator.key-value
//          ^^^^^ storage.type.array
//               ^ punctuation.definition.array.begin
//                 ^ constant.numeric.integer
//                   ^^ keyword.operator.range
//                      ^^ constant.numeric.integer
//                         ^ punctuation.definition.array.end
//                           ^^ keyword.control.of
//                              ^^ punctuation.definition.comment.begin
//                              ^^^^^^^ comment.line.double-slash
            DWORD ;  //integer
// ^^^^^^^^^^^^^^^^^^^^^^^^^^^ meta.block.fc.header meta.block.var.temp
// ^^^^^^^^^^^^^^ meta.definition.variable.storage meta.sequence.array
//          ^^^^^ storage.type.dword
     _ST  : STRUCT  //structure
// ^^^^^^^^^^^^^^^^^^^^^^^^^^^^ meta.block.fc.header meta.block.var.temp
//   ^^^^^ meta.definition.variable - meta.definition.variable.storage
//         ^^^^^^^^^^^^^^^^^^^^ meta.definition.variable.storage
//          ^^^^^^^^^^^^^^^^^^^ meta.struct
//   ^^^ variable.other
//        ^ punctuation.separator.key-value
//          ^^^^^^ storage.type.struct.begin
       RUN : BOOL ;  //bool
// ^^^^^^^^^^^^^^^^^^^^^^^^ meta.block.fc.header meta.block.var.temp meta.definition.variable.storage meta.struct
//     ^^^^^ meta.definition.variable
//          ^^^^^^ meta.definition.variable.storage meta.definition.variable.storage
//     ^^^ variable.other
//         ^ punctuation.separator.key-value
//           ^^^^ storage.type.bool
       ID  : INT  ;  //integer
// ^^^^^^^^^^^^^^^^^^^^^^^^^^^ meta.block.fc.header meta.block.var.temp meta.definition.variable.storage meta.struct
//     ^^^^^ meta.definition.variable
//          ^^^^^^ meta.definition.variable.storage meta.definition.variable.storage
//     ^^ variable.other
//         ^ punctuation.separator.key-value
//           ^^^ storage.type.integer
       _S1  : STRING[32] ;  //string
// ^^^^^^^^^^^^^^^^^^^^^^^^^^^^^^^^^ meta.block.fc.header meta.block.var.temp meta.definition.variable.storage meta.struct
//     ^^^^^ meta.definition.variable
//           ^^^^^^^^^^^^ meta.definition.variable.storage meta.definition.variable.storage
//     ^^^ variable.other
//          ^ punctuation.separator.key-value
//            ^^^^^^^^^^ storage.type.string
    END_STRUCT ;
//^^^^^^^^^^^^^^^ meta.block.fc.header meta.block.var.temp
//^^^^^^^^^^^^^ meta.definition.variable.storage
//^^^^^^^^^^^^ meta.struct
//  ^^^^^^^^^^ storage.type.struct.end
//             ^ punctuation.terminator.statement
     _AS  : ARRAY[ 0 .. 20 ] OF STRUCT //array
// ^^^^^^^^^^^^^^^^^^^^^^^^^^^^^^^^^^^^^^^^^^^ meta.block.fc.header meta.block.var.temp
//   ^^^^^ meta.definition.variable - meta.definition.variable.storage
//         ^^^^^^^^^^^^^^^^^^^^^^^^^^^^^^^^^^^ meta.definition.variable.storage
//          ^^^^^^^^^^^^^^^^^^^^^^^^^^^^^^^^^^ meta.sequence.array
//                              ^^^^^^^^^^^^^^ meta.struct
//   ^^^ variable.other
//        ^ punctuation.separator.key-value
//          ^^^^^ storage.type.array
//               ^ punctuation.definition.array.begin
//                 ^ constant.numeric.integer
//                   ^^ keyword.operator.range
//                      ^^ constant.numeric.integer
//                         ^ punctuation.definition.array.end
//                           ^^ keyword.control.of
//                              ^^^^^^ storage.type.struct.begin
//                                     ^^ punctuation.definition.comment.begin
//                                     ^^^^^^^ comment.line.double-slash
       RUN : BOOL ;  //bool
// ^^^^^^^^^^^^^^^^^^^^^^^^ meta.block.fc.header meta.block.var.temp meta.definition.variable.storage meta.sequence.array meta.struct
//     ^^^^^ meta.definition.variable
//          ^^^^^^ meta.definition.variable.storage meta.definition.variable.storage
//     ^^^ variable.other
//         ^ punctuation.separator.key-value
//           ^^^^ storage.type.bool
       ID  : INT  ;  //integer
// ^^^^^^^^^^^^^^^^^^^^^^^^^^^ meta.block.fc.header meta.block.var.temp meta.definition.variable.storage meta.sequence.array meta.struct
//     ^^^^^ meta.definition.variable
//          ^^^^^^ meta.definition.variable.storage meta.definition.variable.storage
//     ^^ variable.other
//         ^ punctuation.separator.key-value
//           ^^^ storage.type.integer
       _S1  : STRING[32] ;  //string
// ^^^^^^^^^^^^^^^^^^^^^^^^^^^^^^^^^ meta.block.fc.header meta.block.var.temp meta.definition.variable.storage meta.sequence.array meta.struct
//     ^^^^^ meta.definition.variable
//           ^^^^^^^^^^^^ meta.definition.variable.storage meta.definition.variable.storage
//     ^^^ variable.other
//          ^ punctuation.separator.key-value
//            ^^^^^^^^^^ storage.type.string
    END_STRUCT ;
//^^^^^^^^^^^^^^^ meta.block.fc.header meta.block.var.temp
//^^^^^^^^^^^^^ meta.definition.variable.storage
//^^^^^^^^^^^^ meta.struct
//  ^^^^^^^^^^ storage.type.struct.end
//             ^ punctuation.terminator.statement
   END_VAR
// <- meta.block.fc.header meta.block.var.temp
// ^^^^^^^ meta.block.fc.header meta.block.var.temp
// ^^^^^^^ keyword.control.var.end

   VAR
// ^^^ meta.block.fc.header invalid.illegal
   END_VAR
// ^^^^^^^ meta.block.fc.header invalid.illegal

// NOTE: unclosed input declaration context

   VAR_INPUT
// ^^^^^^^^^ keyword.control.var.input.begin.s7.awl

   BEGIN
// <- meta.block.fc.header - meta.block.fc.body
//^ meta.block.fc.header - meta.block.fc.body
// ^^^^^ meta.block.fc.body - meta.block.fc.header
// ^^^^^ keyword.other.begin

   NETWORK //network 1
// <- meta.block.fc.body
// ^^^^^^^^^^^^^^^^^^^ meta.block.fc.body meta.block.network
// ^^^^^^^ keyword.control.network
   TITLE =CALL test
// <- meta.block.fc.body meta.block.network
// ^^^^^^^^^^^^^^^^ meta.block.fc.body meta.block.network
// ^^^^^^^ meta.mapping.key
//        ^^^^^^^^^ meta.mapping.value
// ^^^^^ entity.other.attribute-name.title
//       ^ punctuation.separator.key-value.title
//        ^^^^^^^^^ entity.name.section.s7.awl
///////////////////////////////////////////////////////////////////////////////
// basic operations                                                          //
///////////////////////////////////////////////////////////////////////////////
      BLD  1; // comment
//    ^^^ keyword.operator.nop
//         ^ constant.numeric.integer
//          ^ punctuation.terminator.statement
      NOP  0; // comment
//    ^^^ keyword.operator.nop
//         ^ constant.numeric.integer
//          ^ punctuation.terminator.statement

///////////////////////////////////////////////////////////////////////////////
// datablock operations                                                      //
///////////////////////////////////////////////////////////////////////////////

      AUF   DB 10;
// <- meta.block.fc.body.s7.awl meta.block.network.s7.awl
//^^^^^^^^^^^^^^^^^ meta.block.fc.body.s7.awl meta.block.network.s7.awl
//       ^^^^^^^^^ meta.operand.datablock.s7.awl
//                ^ - meta.operand.datablock.s7.awl
//    ^^^ keyword.operator.load.db.s7.awl
//          ^^^^^ variable.language.db.s7.awl
//               ^ punctuation.terminator.statement.s7.awl
      AUF   DB [MW 10];
// <- meta.block.fc.body.s7.awl meta.block.network.s7.awl
//^^^^^^^^^^^^^^^^^^^^^ meta.block.fc.body.s7.awl meta.block.network.s7.awl
//       ^^^^^^^^^^^^^^ meta.operand.datablock.s7.awl
//                     ^ - meta.operand.datablock.s7.awl
//    ^^^ keyword.operator.load.db.s7.awl
//          ^^^^^^^^^^ variable.language.db.s7.awl
//                    ^ punctuation.terminator.statement.s7.awl
      AUF   "IDB_Block";
// <- meta.block.fc.body.s7.awl meta.block.network.s7.awl
//^^^^^^^^^^^^^^^^^^^^^^^ meta.block.fc.body.s7.awl meta.block.network.s7.awl
//       ^^^^^^^^^^^^^^^ meta.operand.datablock.s7.awl
//                      ^ - meta.operand.datablock.s7.awl
//    ^^^ keyword.operator.load.db.s7.awl
//          ^ string.quoted.double punctuation.definition.string.begin
//          ^^^^^^^^^^^ meta.string
//           ^^^^^^^^^ variable.other.symbol - string
//                    ^ string.quoted.double punctuation.definition.string.end
//                     ^ punctuation.terminator.statement.s7.awl
      AUF   DBNO;
// <- meta.block.fc.body.s7.awl meta.block.network.s7.awl
//^^^^^^^^^^^^^^^^ meta.block.fc.body.s7.awl meta.block.network.s7.awl
//       ^^^^^^^^ meta.operand.datablock.s7.awl
//               ^ - meta.operand.datablock.s7.awl
//    ^^^ keyword.operator.load.db.s7.awl
//          ^^^^ invalid.illegal
//              ^ punctuation.terminator.statement.s7.awl
      AUF   DINO;
// <- meta.block.fc.body.s7.awl meta.block.network.s7.awl
//^^^^^^^^^^^^^^^^ meta.block.fc.body.s7.awl meta.block.network.s7.awl
//       ^^^^^^^^ meta.operand.datablock.s7.awl
//               ^ - meta.operand.datablock.s7.awl
//    ^^^ keyword.operator.load.db.s7.awl
//          ^^^^ invalid.illegal
//              ^ punctuation.terminator.statement.s7.awl
      TDB   ;
// <- meta.block.fc.body.s7.awl meta.block.network.s7.awl
//^^^^^^^^^^^^^^^^ meta.block.fc.body.s7.awl meta.block.network.s7.awl
//    ^^^ keyword.operator.db.s7.awl
//          ^ punctuation.terminator.statement.s7.awl

///////////////////////////////////////////////////////////////////////////////
// logical operations                                                        //
///////////////////////////////////////////////////////////////////////////////

      U     E3.0;
// <- meta.block.fc.body meta.block.network
// ^^^^^^^^^^^^^^^ meta.block.fc.body meta.block.network
//     ^^^^^^^^^^ meta.operand.logical.s7.awl
//    ^ keyword.operator.logical
//          ^^^^ variable.language.address
//            ^ punctuation.separator.decimal
//              ^ punctuation.terminator.statement
//               ^ - invalid
      U     A3.0;
// <- meta.block.fc.body meta.block.network
// ^^^^^^^^^^^^^^^ meta.block.fc.body meta.block.network
//     ^^^^^^^^^^ meta.operand.logical.s7.awl
//    ^ keyword.operator.logical
//          ^^^^ variable.language.address
//            ^ punctuation.separator.decimal
//              ^ punctuation.terminator.statement
//               ^ - invalid
      U     L3.0;
// <- meta.block.fc.body meta.block.network
// ^^^^^^^^^^^^^^^ meta.block.fc.body meta.block.network
//     ^^^^^^^^^^ meta.operand.logical.s7.awl
//    ^ keyword.operator.logical
//          ^^^^ variable.language.address
//            ^ punctuation.separator.decimal
//              ^ punctuation.terminator.statement
//               ^ - invalid
      U     M3.0;
// <- meta.block.fc.body meta.block.network
// ^^^^^^^^^^^^^^^ meta.block.fc.body meta.block.network
//     ^^^^^^^^^^ meta.operand.logical.s7.awl
//    ^ keyword.operator.logical
//          ^^^^ variable.language.address
//            ^ punctuation.separator.decimal
//              ^ punctuation.terminator.statement
//               ^ - invalid
      U     DBX3.0;
// <- meta.block.fc.body meta.block.network
// ^^^^^^^^^^^^^^^^^ meta.block.fc.body meta.block.network
//     ^^^^^^^^^^^^ meta.operand.logical.s7.awl
//    ^ keyword.operator.logical
//          ^^^^^^ variable.language.address
//              ^ punctuation.separator.decimal
//                ^ punctuation.terminator.statement
//                 ^ - invalid
      U     DIX3.0;
// <- meta.block.fc.body meta.block.network
// ^^^^^^^^^^^^^^^^^ meta.block.fc.body meta.block.network
//     ^^^^^^^^^^^^ meta.operand.logical.s7.awl
//    ^ keyword.operator.logical
//          ^^^^^^ variable.language.address
//              ^ punctuation.separator.decimal
//                ^ punctuation.terminator.statement
//                 ^ - invalid
      U     DB10.DBX3.0;
// <- meta.block.fc.body meta.block.network
// ^^^^^^^^^^^^^^^^^^^^^^ meta.block.fc.body meta.block.network
//     ^^^^^^^^^^^^^^^^^ meta.operand.logical.s7.awl
//    ^ keyword.operator.logical
//          ^^^^ variable.language.db
//              ^ punctuation.accessor.dot
//               ^^^^^^ variable.language.address
//                   ^ punctuation.separator.decimal
//                     ^ punctuation.terminator.statement
//                      ^ - invalid

///////////////////////////////////////////////////////////////////////////////
// load values into akku1                                                    //
///////////////////////////////////////////////////////////////////////////////
      L    MB10;  // comment
// <- meta.block.fc.body meta.block.network
// ^^^^^^^^^^^^^^^^^^^^^^^^^ meta.block.fc.body meta.block.network
//    ^ keyword.operator.arithmetic.load
//         ^^^^ variable.language.address
//             ^ punctuation.terminator.statement
//                ^^ punctuation.definition.comment.begin
//                ^^^^^^^^^^ comment.line.double-slash
      L    MB[ LD0 ]; // comment
// <- meta.block.fc.body meta.block.network
// ^^^^^^^^^^^^^^^^^^^^^^^^^^^^ meta.block.fc.body meta.block.network
//         ^^^^^^^^^ meta.operand.numeric
//           ^^^^^^^ meta.brackets
//    ^ keyword.operator.arithmetic.load
//         ^^ variable.language.address
//           ^ punctuation.section.brackets.begin
//             ^^^ variable.language.address
//                 ^ punctuation.section.brackets.end
//                  ^ punctuation.terminator.statement
//                    ^^ punctuation.definition.comment.begin
//                    ^^^^^^^^^^ comment.line.double-slash
      L    MW10;  // comment
// <- meta.block.fc.body meta.block.network
// ^^^^^^^^^^^^^^^^^^^^^^^^^ meta.block.fc.body meta.block.network
//    ^ keyword.operator.arithmetic.load
//         ^^^^ variable.language.address
//             ^ punctuation.terminator.statement
//                ^^ punctuation.definition.comment.begin
//                ^^^^^^^^^^ comment.line.double-slash
      L    MW[ LD0 ]; // comment
// <- meta.block.fc.body meta.block.network
// ^^^^^^^^^^^^^^^^^^^^^^^^^^^^ meta.block.fc.body meta.block.network
//         ^^^^^^^^^ meta.operand.numeric
//           ^^^^^^^ meta.brackets
//    ^ keyword.operator.arithmetic.load
//         ^^ variable.language.address
//           ^ punctuation.section.brackets.begin
//             ^^^ variable.language.address
//                 ^ punctuation.section.brackets.end
//                  ^ punctuation.terminator.statement
//                    ^^ punctuation.definition.comment.begin
//                    ^^^^^^^^^^ comment.line.double-slash
      L    MD10;  // comment
// <- meta.block.fc.body meta.block.network
// ^^^^^^^^^^^^^^^^^^^^^^^^^ meta.block.fc.body meta.block.network
//    ^ keyword.operator.arithmetic.load
//         ^^^^ variable.language.address
//             ^ punctuation.terminator.statement
//                ^^ punctuation.definition.comment.begin
//                ^^^^^^^^^^ comment.line.double-slash
      L    MD[ LD0 ]; // comment
// <- meta.block.fc.body meta.block.network
// ^^^^^^^^^^^^^^^^^^^^^^^^^^^^ meta.block.fc.body meta.block.network
//         ^^^^^^^^^ meta.operand.numeric
//           ^^^^^^^ meta.brackets
//    ^ keyword.operator.arithmetic.load
//         ^^ variable.language.address
//           ^ punctuation.section.brackets.begin
//             ^^^ variable.language.address
//                 ^ punctuation.section.brackets.end
//                  ^ punctuation.terminator.statement
//                    ^^ punctuation.definition.comment.begin
//                    ^^^^^^^^^^ comment.line.double-slash
      L    M10.0;  // comment
// <- meta.block.fc.body meta.block.network
// ^^^^^^^^^^^^^^^^^^^^^^^^^^ meta.block.fc.body meta.block.network
//    ^ keyword.operator.arithmetic.load
//         ^^^^^ invalid.illegal
//              ^ punctuation.terminator.statement
//                 ^^ punctuation.definition.comment.begin
//                 ^^^^^^^^^^ comment.line.double-slash
      L    LB10;  // comment
// <- meta.block.fc.body meta.block.network
// ^^^^^^^^^^^^^^^^^^^^^^^^^ meta.block.fc.body meta.block.network
//    ^ keyword.operator.arithmetic.load
//         ^^^^ variable.language.address
//             ^ punctuation.terminator.statement
//                ^^ punctuation.definition.comment.begin
//                ^^^^^^^^^^ comment.line.double-slash
      L    LB[ LD0 ]; // comment
// <- meta.block.fc.body meta.block.network
// ^^^^^^^^^^^^^^^^^^^^^^^^^^^^ meta.block.fc.body meta.block.network
//         ^^^^^^^^^ meta.operand.numeric
//           ^^^^^^^ meta.brackets
//    ^ keyword.operator.arithmetic.load
//         ^^ variable.language.address
//           ^ punctuation.section.brackets.begin
//             ^^^ variable.language.address
//                 ^ punctuation.section.brackets.end
//                  ^ punctuation.terminator.statement
//                    ^^ punctuation.definition.comment.begin
//                    ^^^^^^^^^^ comment.line.double-slash
      L    LW10;  // comment
// <- meta.block.fc.body meta.block.network
// ^^^^^^^^^^^^^^^^^^^^^^^^^ meta.block.fc.body meta.block.network
//    ^ keyword.operator.arithmetic.load
//         ^^^^ variable.language.address
//             ^ punctuation.terminator.statement
//                ^^ punctuation.definition.comment.begin
//                ^^^^^^^^^^ comment.line.double-slash
      L    LW[ LD0 ]; // comment
// <- meta.block.fc.body meta.block.network
// ^^^^^^^^^^^^^^^^^^^^^^^^^^^^ meta.block.fc.body meta.block.network
//         ^^^^^^^^^ meta.operand.numeric
//           ^^^^^^^ meta.brackets
//    ^ keyword.operator.arithmetic.load
//         ^^ variable.language.address
//           ^ punctuation.section.brackets.begin
//             ^^^ variable.language.address
//                 ^ punctuation.section.brackets.end
//                  ^ punctuation.terminator.statement
//                    ^^ punctuation.definition.comment.begin
//                    ^^^^^^^^^^ comment.line.double-slash
      L    LD10;  // comment
// <- meta.block.fc.body meta.block.network
// ^^^^^^^^^^^^^^^^^^^^^^^^^ meta.block.fc.body meta.block.network
//    ^ keyword.operator.arithmetic.load
//         ^^^^ variable.language.address
//             ^ punctuation.terminator.statement
//                ^^ punctuation.definition.comment.begin
//                ^^^^^^^^^^ comment.line.double-slash
      L    LD[ LD0 ]; // comment
// <- meta.block.fc.body meta.block.network
// ^^^^^^^^^^^^^^^^^^^^^^^^^^^^ meta.block.fc.body meta.block.network
//         ^^^^^^^^^ meta.operand.numeric
//           ^^^^^^^ meta.brackets
//    ^ keyword.operator.arithmetic.load
//         ^^ variable.language.address
//           ^ punctuation.section.brackets.begin
//             ^^^ variable.language.address
//                 ^ punctuation.section.brackets.end
//                  ^ punctuation.terminator.statement
//                    ^^ punctuation.definition.comment.begin
//                    ^^^^^^^^^^ comment.line.double-slash
      L    L10.0;  // comment
// <- meta.block.fc.body meta.block.network
// ^^^^^^^^^^^^^^^^^^^^^^^^^^ meta.block.fc.body meta.block.network
//    ^ keyword.operator.arithmetic.load
//         ^^^^^ invalid.illegal
//              ^ punctuation.terminator.statement
//                 ^^ punctuation.definition.comment.begin
//                 ^^^^^^^^^^ comment.line.double-slash
      L     T 10;  // comment
// <- meta.block.fc.body meta.block.network
// ^^^^^^^^^^^^^^^^^^^^^^^^^^ meta.block.fc.body meta.block.network
//    ^ keyword.operator.arithmetic.load
//          ^^^^ variable.language.timer
//              ^ punctuation.terminator.statement
//                 ^^ punctuation.definition.comment.begin
//                 ^^^^^^^^^^ comment.line.double-slash
      L     T [MW10];  // comment
// <- meta.block.fc.body meta.block.network
// ^^^^^^^^^^^^^^^^^^^^^^^^^^^^^ meta.block.fc.body meta.block.network
//    ^ keyword.operator.arithmetic.load
//          ^^^^^^^^ variable.language.timer
//            ^^^^^^ meta.brackets
//            ^ punctuation.section.brackets.begin
//             ^^^^ variable.language.address
//                 ^ punctuation.section.brackets.end
//                  ^ punctuation.terminator.statement
//                     ^^ punctuation.definition.comment.begin
//                     ^^^^^^^^^^ comment.line.double-slash
      L     Z 10;  // comment
// <- meta.block.fc.body meta.block.network
// ^^^^^^^^^^^^^^^^^^^^^^^^^^ meta.block.fc.body meta.block.network
//    ^ keyword.operator.arithmetic.load
//          ^^^^ variable.language.counter
//              ^ punctuation.terminator.statement
//                 ^^ punctuation.definition.comment.begin
//                 ^^^^^^^^^^ comment.line.double-slash
      L     Z [MW10];  // comment
// <- meta.block.fc.body meta.block.network
// ^^^^^^^^^^^^^^^^^^^^^^^^^^^^^ meta.block.fc.body meta.block.network
//    ^ keyword.operator.arithmetic.load
//          ^^^^^^^^ variable.language.counter
//            ^^^^^^ meta.brackets
//            ^ punctuation.section.brackets.begin
//             ^^^^ variable.language.address
//                 ^ punctuation.section.brackets.end
//                  ^ punctuation.terminator.statement
//                     ^^ punctuation.definition.comment.begin
//                     ^^^^^^^^^^ comment.line.double-slash
      L     DBNO;  // comment
// <- meta.block.fc.body meta.block.network
// ^^^^^^^^^^^^^^^^^^^^^^^^^^ meta.block.fc.body meta.block.network
//    ^ keyword.operator.arithmetic.load
//          ^^^^ variable.language
//              ^ punctuation.terminator.statement
//                 ^^ punctuation.definition.comment.begin
//                 ^^^^^^^^^^ comment.line.double-slash
      L     DINO;  // comment
// <- meta.block.fc.body meta.block.network
// ^^^^^^^^^^^^^^^^^^^^^^^^^^ meta.block.fc.body meta.block.network
//    ^ keyword.operator.arithmetic.load
//          ^^^^ variable.language
//              ^ punctuation.terminator.statement
//                 ^^ punctuation.definition.comment.begin
//                 ^^^^^^^^^^ comment.line.double-slash
      L     DBB  140;  // comment
// <- meta.block.fc.body meta.block.network
// ^^^^^^^^^^^^^^^^^^^^^^^^^^^^^^ meta.block.fc.body meta.block.network
//    ^ keyword.operator.arithmetic.load
//          ^^^^^^^^ variable.language.address.s7.awl
//                  ^ punctuation.terminator.statement
//                     ^^ punctuation.definition.comment.begin
//                     ^^^^^^^^^^ comment.line.double-slash
      L     DBW  140;  // comment
// <- meta.block.fc.body meta.block.network
// ^^^^^^^^^^^^^^^^^^^^^^^^^^^^^^ meta.block.fc.body meta.block.network
//    ^ keyword.operator.arithmetic.load
//          ^^^^^^^^ variable.language.address.s7.awl
//                  ^ punctuation.terminator.statement
//                     ^^ punctuation.definition.comment.begin
//                     ^^^^^^^^^^ comment.line.double-slash
      L     DBD  140;  // comment
// <- meta.block.fc.body meta.block.network
// ^^^^^^^^^^^^^^^^^^^^^^^^^^^^^^ meta.block.fc.body meta.block.network
//    ^ keyword.operator.arithmetic.load
//          ^^^^^^^^ variable.language.address.s7.awl
//                  ^ punctuation.terminator.statement
//                     ^^ punctuation.definition.comment.begin
//                     ^^^^^^^^^^ comment.line.double-slash
      L     DIB  140;  // comment
// <- meta.block.fc.body meta.block.network
// ^^^^^^^^^^^^^^^^^^^^^^^^^^^^^^ meta.block.fc.body meta.block.network
//    ^ keyword.operator.arithmetic.load
//          ^^^^^^^^ variable.language.address.s7.awl
//                  ^ punctuation.terminator.statement
//                     ^^ punctuation.definition.comment.begin
//                     ^^^^^^^^^^ comment.line.double-slash
      L     DIW  140;  // comment
// <- meta.block.fc.body meta.block.network
// ^^^^^^^^^^^^^^^^^^^^^^^^^^^^^^ meta.block.fc.body meta.block.network
//    ^ keyword.operator.arithmetic.load
//          ^^^^^^^^ variable.language.address.s7.awl
//                  ^ punctuation.terminator.statement
//                     ^^ punctuation.definition.comment.begin
//                     ^^^^^^^^^^ comment.line.double-slash
      L     DID  140;  // comment
// <- meta.block.fc.body meta.block.network
// ^^^^^^^^^^^^^^^^^^^^^^^^^^^^^^ meta.block.fc.body meta.block.network
//    ^ keyword.operator.arithmetic.load
//          ^^^^^^^^ variable.language.address.s7.awl
//                  ^ punctuation.terminator.statement
//                     ^^ punctuation.definition.comment.begin
//                     ^^^^^^^^^^ comment.line.double-slash
      L    DB200.DBB20;  // comment
// <- meta.block.fc.body meta.block.network
// ^^^^^^^^^^^^^^^^^^^^^^^^^^^^^^^^ meta.block.fc.body meta.block.network
//    ^ keyword.operator.arithmetic.load
//         ^^^^^ variable.language.db
//              ^ punctuation.accessor.dot
//               ^^^^^ variable.language.address
//                    ^ punctuation.terminator.statement
//                       ^^ punctuation.definition.comment.begin
//                       ^^^^^^^^^^ comment.line.double-slash
      L    DB200.DBW20;  // comment
// <- meta.block.fc.body meta.block.network
// ^^^^^^^^^^^^^^^^^^^^^^^^^^^^^^^^ meta.block.fc.body meta.block.network
//    ^ keyword.operator.arithmetic.load
//         ^^^^^ variable.language.db
//              ^ punctuation.accessor.dot
//               ^^^^^ variable.language.address
//                    ^ punctuation.terminator.statement
//                       ^^ punctuation.definition.comment.begin
//                       ^^^^^^^^^^ comment.line.double-slash
      L    DB200.DBD20;  // comment
// <- meta.block.fc.body meta.block.network
// ^^^^^^^^^^^^^^^^^^^^^^^^^^^^^^^^ meta.block.fc.body meta.block.network
//    ^ keyword.operator.arithmetic.load
//         ^^^^^ variable.language.db
//              ^ punctuation.accessor.dot
//               ^^^^^ variable.language.address
//                    ^ punctuation.terminator.statement
//                       ^^ punctuation.definition.comment.begin
//                       ^^^^^^^^^^ comment.line.double-slash
      L    DB200.DBX20.0;  // comment
// <- meta.block.fc.body meta.block.network
// ^^^^^^^^^^^^^^^^^^^^^^^^^^^^^^^^^^ meta.block.fc.body meta.block.network
//    ^ keyword.operator.arithmetic.load
//         ^^^^^^^^^^^^^ invalid.illegal
//                      ^ punctuation.terminator.statement
//                         ^^ punctuation.definition.comment.begin
//                         ^^^^^^^^^^ comment.line.double-slash
      L    "datablock".struct[ 4 ].value;  // comment
// <- meta.block.fc.body meta.block.network
// ^^^^^^^^^^^^^^^^^^^^^^^^^^^^^^^^^^^^^^^^^^^^^ meta.block.fc.body meta.block.network
//    ^ keyword.operator.arithmetic.load
//         ^ string.quoted.double punctuation.definition.string.begin - variable
//         ^^^^^^^^^^^ meta.string
//          ^^^^^^^^^ variable.other.symbol - string
//                   ^ string.quoted.double punctuation.definition.string.end - variable
//                    ^ punctuation.accessor.dot
//                     ^^^^^^ variable.other.member
//                           ^ punctuation.section.brackets.begin
//                           ^^^^^ meta.brackets
//                             ^ constant.numeric.integer
//                               ^ punctuation.section.brackets.end
//                                ^ punctuation.accessor.dot
//                                 ^^^^^ variable.other.member
//                                      ^ punctuation.terminator.statement
//                                         ^^ punctuation.definition.comment.begin
//                                         ^^^^^^^^^^ comment.line.double-slash
      L    "datablock".struct.value;  // comment
// <- meta.block.fc.body meta.block.network
// ^^^^^^^^^^^^^^^^^^^^^^^^^^^^^^^^^^^^^^^^^^^^^ meta.block.fc.body meta.block.network
//    ^ keyword.operator.arithmetic.load
//         ^ string.quoted.double punctuation.definition.string.begin - variable
//         ^^^^^^^^^^^ meta.string
//          ^^^^^^^^^ variable.other.symbol - string
//                   ^ string.quoted.double punctuation.definition.string.end - variable
//                    ^ punctuation.accessor.dot
//                     ^^^^^^ variable.other.member
//                           ^ punctuation.accessor.dot
//                            ^^^^^ variable.other.member
//                                 ^ punctuation.terminator.statement
//                                    ^^ punctuation.definition.comment.begin
//                                    ^^^^^^^^^^ comment.line.double-slash
      L    #local[1].array[0].value[ 10 ];  // comment
// <- meta.block.fc.body meta.block.network
// ^^^^^^^^^^^^^^^^^^^^^^^^^^^^^^^^^^^^^^^^^^^^^^ meta.block.fc.body meta.block.network
//    ^ keyword.operator.arithmetic.load
//         ^ punctuation.definition.variable.begin
//          ^^^^^ variable.other.local
//               ^ punctuation.section.brackets.begin
//               ^^^ meta.brackets
//                ^ constant.numeric.integer
//                 ^ punctuation.section.brackets.end
//                  ^ punctuation.accessor.dot
//                   ^^^^^ variable.other.member
//                        ^ punctuation.section.brackets.begin
//                        ^^^ meta.brackets
//                         ^ constant.numeric.integer
//                          ^ punctuation.section.brackets.end
//                           ^ punctuation.accessor.dot
//                            ^^^^^ variable.other.member
//                                 ^ punctuation.section.brackets.begin
//                                 ^^^^^^ meta.brackets
//                                   ^^ constant.numeric.integer
//                                      ^ punctuation.section.brackets.end
//                                       ^ punctuation.terminator.statement
//                                          ^^ punctuation.definition.comment.begin
//                                          ^^^^^^^^^^ comment.line.double-slash
      L    P# P0.0; // comment
// <- meta.block.fc.body meta.block.network
// ^^^^^^^^^^^^^^^^^^^^^^^^^^^^^ meta.block.fc.body meta.block.network
//    ^ keyword.operator.arithmetic.load
//         ^^ storage.type.numeric.s7.awl
//         ^^^^^^^ constant.language.pointer
//              ^ punctuation.separator.decimal.s7.awl
//                ^ punctuation.terminator.statement
//                  ^^ punctuation.definition.comment.begin
//                  ^^^^^^^^^^ comment.line.double-slash
      L    P##local;  // comment
// <- meta.block.fc.body meta.block.network
// ^^^^^^^^^^^^^^^^^^^^^^^^^^^^^ meta.block.fc.body meta.block.network
//    ^ keyword.operator.arithmetic.load
//         ^^ storage.type.numeric.s7.awl
//           ^ punctuation.definition.variable.begin
//            ^^^^^ variable.other.local
//                 ^ punctuation.terminator.statement
//                    ^^ punctuation.definition.comment.begin
//                    ^^^^^^^^^^ comment.line.double-slash
      L    P#120.4;  // comment
// <- meta.block.fc.body meta.block.network
// ^^^^^^^^^^^^^^^^^^^^^^^^^^^^^ meta.block.fc.body meta.block.network
//    ^ keyword.operator.arithmetic.load
//         ^^ storage.type.numeric.s7.awl
//         ^^^^^^^ constant.language.pointer
//                ^ punctuation.terminator.statement
//                   ^^ punctuation.definition.comment.begin
//                   ^^^^^^^^^^ comment.line.double-slash
      L    P#DBX120.4;  // comment
// <- meta.block.fc.body meta.block.network
// ^^^^^^^^^^^^^^^^^^^^^^^^^^^^^^^ meta.block.fc.body meta.block.network
//    ^ keyword.operator.arithmetic.load
//         ^^ storage.type.numeric.s7.awl
//         ^^^^^^^^^^ constant.language.pointer
//                 ^ punctuation.separator.decimal
//                   ^ punctuation.terminator.statement
//                      ^^ punctuation.definition.comment.begin
//                      ^^^^^^^^^^ comment.line.double-slash
      L    P#DB2.DBX120.4;  // comment
// <- meta.block.fc.body meta.block.network
// ^^^^^^^^^^^^^^^^^^^^^^^^^^^^^^^^^^^^ meta.block.fc.body meta.block.network
//    ^ keyword.operator.arithmetic.load
//         ^^ storage.type.numeric.s7.awl
//         ^^^^^^^^^^^^^^ constant.language.pointer
//              ^ punctuation.accessor.dot
//                     ^ punctuation.separator.decimal
//                       ^ punctuation.terminator.statement
//                          ^^ punctuation.definition.comment.begin
//                          ^^^^^^^^^^ comment.line.double-slash
      L    2#0000_0000_0000_0000_0000_0000_0000_0000 ;
// <- meta.block.fc.body meta.block.network
// ^^^^^^^^^^^^^^^^^^^^^^^^^^^^^^^^^^^^^^^^^^^^^^^^^^^^ meta.block.fc.body meta.block.network
//    ^ keyword.operator.arithmetic.load
//         ^^ storage.type.numeric.s7.awl
//         ^^^^^^^^^^^^^^^^^^^^^^^^^^^^^^^^^^^^^^^^^ constant.numeric.bin
//               ^ punctuation.separator.bin
//                    ^ punctuation.separator.bin
//                         ^ punctuation.separator.bin
//                              ^ punctuation.separator.bin
//                                   ^ punctuation.separator.bin
//                                        ^ punctuation.separator.bin
//                                             ^ punctuation.separator.bin
//                                                  ^ - invalid
//                                                   ^ punctuation.terminator.statement
//                                                    ^ - invalid
      L    2#1111_1111_1111_1111_1111_1111_1111_1111 ;
// <- meta.block.fc.body meta.block.network
// ^^^^^^^^^^^^^^^^^^^^^^^^^^^^^^^^^^^^^^^^^^^^^^^^^^^^ meta.block.fc.body meta.block.network
//    ^ keyword.operator.arithmetic.load
//         ^^ storage.type.numeric.s7.awl
//         ^^^^^^^^^^^^^^^^^^^^^^^^^^^^^^^^^^^^^^^^^ constant.numeric.bin
//               ^ punctuation.separator.bin
//                    ^ punctuation.separator.bin
//                         ^ punctuation.separator.bin
//                              ^ punctuation.separator.bin
//                                   ^ punctuation.separator.bin
//                                        ^ punctuation.separator.bin
//                                             ^ punctuation.separator.bin
//                                                  ^ - invalid
//                                                   ^ punctuation.terminator.statement
//                                                    ^ - invalid
      L    2#1121_1111_1A11_1111_111_11011_1111_1111 ;
// <- meta.block.fc.body meta.block.network
// ^^^^^^^^^^^^^^^^^^^^^^^^^^^^^^^^^^^^^^^^^^^^^^^^^^^^ meta.block.fc.body meta.block.network
//    ^ keyword.operator.arithmetic.load
//         ^^ storage.type.numeric.s7.awl
//         ^^^^^^^^^^^^^^^^^^^^^^^^^^^^^^^^^^^^^^^^^ constant.numeric.bin
//             ^ invalid.illegal.bin
//               ^ punctuation.separator.bin
//                    ^ punctuation.separator.bin
//                      ^ invalid.illegal.bin
//                         ^ punctuation.separator.bin
//                              ^ punctuation.separator.bin
//                                  ^ punctuation.separator.bin
//                                        ^ punctuation.separator.bin
//                                             ^ punctuation.separator.bin
//                                                  ^ - invalid
//                                                   ^ punctuation.terminator.statement
//                                                    ^ - invalid
      L    B#16#0 ;
// <- meta.block.fc.body meta.block.network
// ^^^^^^^^^^^^^^^^^ meta.block.fc.body meta.block.network
//    ^ keyword.operator.arithmetic.load
//         ^^ storage.type.numeric.s7.awl
//         ^^^^^^ constant.numeric.integer.hexadecimal
//               ^ - invalid
//                ^ punctuation.terminator.statement
//                 ^ - invalid
      L    byte#16#0 ;
// <- meta.block.fc.body meta.block.network
// ^^^^^^^^^^^^^^^^^^^^ meta.block.fc.body meta.block.network
//    ^ keyword.operator.arithmetic.load
//         ^^^^^ storage.type.numeric.s7.awl
//         ^^^^^^^^^ constant.numeric.integer.hexadecimal
//                  ^ - invalid
//                   ^ punctuation.terminator.statement
//                    ^ - invalid
      L    W#16#0 ;
// <- meta.block.fc.body meta.block.network
// ^^^^^^^^^^^^^^^^^ meta.block.fc.body meta.block.network
//    ^ keyword.operator.arithmetic.load
//         ^^ storage.type.numeric.s7.awl
//         ^^^^^^ constant.numeric.integer.hexadecimal
//               ^ - invalid
//                ^ punctuation.terminator.statement
//                 ^ - invalid
      L    word#16#0 ;
// <- meta.block.fc.body meta.block.network
// ^^^^^^^^^^^^^^^^^^^^ meta.block.fc.body meta.block.network
//    ^ keyword.operator.arithmetic.load
//         ^^^^^ storage.type.numeric.s7.awl
//         ^^^^^^^^^ constant.numeric.integer.hexadecimal
//                  ^ - invalid
//                   ^ punctuation.terminator.statement
//                    ^ - invalid
      L    DW#16#0 ;
// <- meta.block.fc.body meta.block.network
// ^^^^^^^^^^^^^^^^^^ meta.block.fc.body meta.block.network
//    ^ keyword.operator.arithmetic.load
//         ^^^ storage.type.numeric.s7.awl
//         ^^^^^^^ constant.numeric.integer.hexadecimal
//                ^ - invalid
//                 ^ punctuation.terminator.statement
//                  ^ - invalid
      L    dword#16#0 ;
// <- meta.block.fc.body meta.block.network
// ^^^^^^^^^^^^^^^^^^^^^ meta.block.fc.body meta.block.network
//    ^ keyword.operator.arithmetic.load
//         ^^^^^^ storage.type.numeric.s7.awl
//         ^^^^^^^^^^ constant.numeric.integer.hexadecimal
//                   ^ - invalid
//                    ^ punctuation.terminator.statement
//                     ^ - invalid
      L    L#16 ;
// <- meta.block.fc.body meta.block.network
// ^^^^^^^^^^^^^^^ meta.block.fc.body meta.block.network
//    ^ keyword.operator.arithmetic.load
//         ^^ storage.type.numeric.s7.awl
//         ^^^^ constant.numeric.integer
//             ^ - invalid
//              ^ punctuation.terminator.statement
//               ^ - invalid
      L    L#-16 ;
// <- meta.block.fc.body meta.block.network
// ^^^^^^^^^^^^^^^ meta.block.fc.body meta.block.network
//    ^ keyword.operator.arithmetic.load
//         ^^ storage.type.numeric.s7.awl
//         ^^^^^ constant.numeric.integer
//              ^ - invalid
//               ^ punctuation.terminator.statement
//                ^ - invalid
      L    2.0323e+002 ;
// <- meta.block.fc.body meta.block.network
// ^^^^^^^^^^^^^^^^^^^^^^ meta.block.fc.body meta.block.network
//    ^ keyword.operator.arithmetic.load
//         ^^^^^^^^^^^ constant.numeric.float
//          ^ punctuation.separator.decimal
//                    ^ - invalid
//                     ^ punctuation.terminator.statement
//                      ^ - invalid
      L    -2.0323e-002 ;
// <- meta.block.fc.body meta.block.network
// ^^^^^^^^^^^^^^^^^^^^^^ meta.block.fc.body meta.block.network
//    ^ keyword.operator.arithmetic.load
//         ^^^^^^^^^^^ constant.numeric.float
//           ^ punctuation.separator.decimal
//                     ^ - invalid
//                      ^ punctuation.terminator.statement
//                       ^ - invalid
      L    C#200 ;
// <- meta.block.fc.body meta.block.network
// ^^^^^^^^^^^^^^^^ meta.block.fc.body meta.block.network
//    ^ keyword.operator.arithmetic.load
//         ^^ storage.type.numeric.s7.awl
//         ^^^^^ constant.numeric.integer.decimal
//              ^ - invalid
//               ^ punctuation.terminator.statement
//                ^ - invalid
      L     S5T#50MS ;
// <- meta.block.fc.body meta.block.network
// ^^^^^^^^^^^^^^^^^^^ meta.block.fc.body meta.block.network
//    ^ keyword.operator.arithmetic.load
//          ^^^^ storage.type.numeric.s7.awl
//          ^^^^^^^^ constant.language.s5time
//              ^^^^ constant.language.time.millisecond
//                  ^ - invalid
//                   ^ punctuation.terminator.statement
//                    ^ - invalid
      L     S5T#50S ;
// <- meta.block.fc.body meta.block.network
// ^^^^^^^^^^^^^^^^^^ meta.block.fc.body meta.block.network
//    ^ keyword.operator.arithmetic.load
//          ^^^^ storage.type.numeric.s7.awl
//          ^^^^^^^ constant.language.s5time
//              ^^^ constant.language.time.second
//                 ^ - invalid
//                  ^ punctuation.terminator.statement
//                   ^ - invalid
      L     S5T#50M ; //Lade 3000s Sekunden
// <- meta.block.fc.body meta.block.network
// ^^^^^^^^^^^^^^^^^^ meta.block.fc.body meta.block.network
//    ^ keyword.operator.arithmetic.load
//          ^^^^ storage.type.numeric.s7.awl
//          ^^^^^^^ constant.language.s5time
//              ^^^ constant.language.time.minute
//                 ^ - invalid
//                  ^ punctuation.terminator.statement
//                   ^ - invalid
//                    ^^^^^^^^^^^^^^^^^^^^^ comment.line
      L     S5T#1H ;
// <- meta.block.fc.body meta.block.network
// ^^^^^^^^^^^^^^^^^ meta.block.fc.body meta.block.network
//    ^ keyword.operator.arithmetic.load
//          ^^^^ storage.type.numeric.s7.awl
//          ^^^^^^ constant.language.s5time
//              ^^ constant.language.time.hour
//                ^ - invalid
//                 ^ punctuation.terminator.statement
//                  ^ - invalid
      L    S5T#2H_30M_58S_200MS ;
// <- meta.block.fc.body meta.block.network
// ^^^^^^^^^^^^^^^^^^^^^^^^^^^^^^^ meta.block.fc.body meta.block.network
//    ^ keyword.operator.arithmetic.load
//         ^^^^^^^^^^^^^^^^^^^^ constant.language.s5time
//         ^^^^ storage.type.numeric.s7.awl
//             ^^ constant.language.time.hour
//               ^ punctuation.separator.time
//                ^^^ constant.language.time.minute
//                   ^ punctuation.separator.time
//                    ^^^ constant.language.time.second
//                       ^ punctuation.separator.time
//                        ^^^^^ constant.language.time.millisecond
//                             ^ - invalid
//                              ^ punctuation.terminator.statement
//                               ^ - invalid
      L    S5T#2H_70M_58S_200MS ;
// <- meta.block.fc.body meta.block.network
// ^^^^^^^^^^^^^^^^^^^^^^^^^^^^^^^ meta.block.fc.body meta.block.network
//    ^ keyword.operator.arithmetic.load
//         ^^^^ storage.type.numeric.s7.awl
//         ^^^^^^^^^^^^^^^^^^^^ constant.language.s5time
//              ^ keyword.other.unit.s7.awl
//                ^^^ invalid.illegal.time
//                      ^ keyword.other.unit.s7.awl
//                           ^^ keyword.other.unit.s7.awl
//                             ^ - invalid
//                              ^ punctuation.terminator.statement
//                               ^ - invalid
      L     T#50MS ;
// <- meta.block.fc.body meta.block.network
// ^^^^^^^^^^^^^^^^^ meta.block.fc.body meta.block.network
//    ^ keyword.operator.arithmetic.load
//          ^^ storage.type.numeric.s7.awl
//          ^^^^^^ constant.language.iec-time
//            ^^^^ constant.language.time.millisecond
//              ^^ keyword.other.unit.s7.awl
//                ^ - invalid
//                 ^ punctuation.terminator.statement
//                  ^ - invalid
      L     T#50S ;
// <- meta.block.fc.body meta.block.network
// ^^^^^^^^^^^^^^^^^ meta.block.fc.body meta.block.network
//    ^ keyword.operator.arithmetic.load
//          ^^ storage.type.numeric.s7.awl
//          ^^^^^ constant.language.iec-time
//            ^^^ constant.language.time.second
//              ^ keyword.other.unit.s7.awl
//               ^ - invalid
//                ^ punctuation.terminator.statement
//                 ^ - invalid
      L     T#50M ;
// <- meta.block.fc.body meta.block.network
// ^^^^^^^^^^^^^^^^^ meta.block.fc.body meta.block.network
//    ^ keyword.operator.arithmetic.load
//          ^^ storage.type.numeric.s7.awl
//          ^^^^^ constant.language.iec-time
//            ^^^ constant.language.time.minute
//              ^ keyword.other.unit.s7.awl
//               ^ - invalid
//                ^ punctuation.terminator.statement
//                 ^ - invalid
      L     T#1H ;
// <- meta.block.fc.body meta.block.network
// ^^^^^^^^^^^^^^^^ meta.block.fc.body meta.block.network
//    ^ keyword.operator.arithmetic.load
//          ^^ storage.type.numeric.s7.awl
//          ^^^^ constant.language.iec-time
//            ^^ constant.language.time.hour
//             ^ keyword.other.unit.s7.awl
//              ^ - invalid
//               ^ punctuation.terminator.statement
//                ^ - invalid
      L     T#2D ;
// <- meta.block.fc.body meta.block.network
// ^^^^^^^^^^^^^^^^ meta.block.fc.body meta.block.network
//    ^ keyword.operator.arithmetic.load
//          ^^ storage.type.numeric.s7.awl
//          ^^^^ constant.language.iec-time
//            ^^ constant.language.time.day
//             ^ keyword.other.unit.s7.awl
//              ^ - invalid
//               ^ punctuation.terminator.statement
//                ^ - invalid
      L    T#24D_23H_59M_59S_999MS ;
// <- meta.block.fc.body meta.block.network
// ^^^^^^^^^^^^^^^^^^^^^^^^^^^^^^^^^^ meta.block.fc.body meta.block.network
//    ^ keyword.operator.arithmetic.load
//         ^^^^^^^^^^^^^^^^^^^^^^^ constant.language.iec-time
//         ^^ storage.type.numeric.s7.awl
//           ^^^ constant.language.time.day
//              ^ punctuation.separator.time
//               ^^^ constant.language.time.hour
//                  ^ punctuation.separator.time
//                   ^^^ constant.language.time.minute
//                      ^ punctuation.separator.time
//                       ^^^ constant.language.time.second
//                          ^ punctuation.separator.time
//                           ^^^^^ constant.language.time.millisecond
//                                ^ - invalid
//                                 ^ punctuation.terminator.statement
//                                  ^ - invalid
      L    T#25D_23H_69M_59S_999MS ;
// <- meta.block.fc.body meta.block.network
// ^^^^^^^^^^^^^^^^^^^^^^^^^^^^^^^^^^ meta.block.fc.body meta.block.network
//    ^ keyword.operator.arithmetic.load
//         ^^^^^^^^^^^^^^^^^^^^^^^ constant.language.iec-time
//         ^^ storage.type.numeric.s7.awl
//           ^^^ invalid.illegal.time.day
//              ^ punctuation.separator.time
//               ^^^ constant.language.time.hour
//                  ^ punctuation.separator.time
//                   ^^^ invalid.illegal.time.minute
//                      ^ punctuation.separator.time
//                       ^^^ constant.language.time.second
//                          ^ punctuation.separator.time
//                           ^^^^^ constant.language.time.millisecond
//                                ^ - invalid
//                                 ^ punctuation.terminator.statement
//                                  ^ - invalid
      L    T#24D_23M_59M_20H_999MS ;
// <- meta.block.fc.body meta.block.network
// ^^^^^^^^^^^^^^^^^^^^^^^^^^^^^^^^^^ meta.block.fc.body meta.block.network
//    ^ keyword.operator.arithmetic.load
//         ^^^^^^^^^^^^^^^^^^^^^^^ constant.language.iec-time
//         ^^ storage.type.numeric.s7.awl
//           ^^^ constant.language.time.day
//              ^ punctuation.separator.time
//               ^^^ invalid.illegal.time.hour
//                  ^ punctuation.separator.time
//                   ^^^ constant.language.time.minute
//                      ^ punctuation.separator.time
//                       ^^^ invalid.illegal.time.second
//                          ^ punctuation.separator.time
//                           ^^^^^ constant.language.time.millisecond
//                                ^ - invalid
//                                 ^ punctuation.terminator.statement
//                                  ^ - invalid
      L    D#2017-12-30 ;
// <- meta.block.fc.body meta.block.network
// ^^^^^^^^^^^^^^^^^^^^^^^ meta.block.fc.body meta.block.network
//    ^ keyword.operator.arithmetic.load
//         ^^ storage.type.numeric.s7.awl
//         ^^^^^^^^^^^^ constant.language.date
//               ^ punctuation.separator.date
//                  ^ punctuation.separator.date
//                     ^ - invalid
//                      ^ punctuation.terminator.statement
//                       ^ - invalid
      L    DATE#2017-12-30 ;
// <- meta.block.fc.body meta.block.network
// ^^^^^^^^^^^^^^^^^^^^^^^^^^ meta.block.fc.body meta.block.network
//    ^ keyword.operator.arithmetic.load
//         ^^^^^ storage.type.numeric.s7.awl
//         ^^^^^^^^^^^^^^^ constant.language.date
//                  ^ punctuation.separator.date
//                     ^ punctuation.separator.date
//                        ^ - invalid
//                         ^ punctuation.terminator.statement
//                          ^ - invalid
      L    TOD#23:59:59.999 ;
// <- meta.block.fc.body meta.block.network
// ^^^^^^^^^^^^^^^^^^^^^^^^^^^ meta.block.fc.body meta.block.network
//    ^ keyword.operator.arithmetic.load
//         ^^^^ storage.type.numeric.s7.awl
//         ^^^^^^^^^^^^^^^^ constant.language.time-of-day
//               ^ punctuation.separator.time
//                  ^ punctuation.separator.time
//                     ^ punctuation.separator.time
//                         ^ - invalid
//                          ^ punctuation.terminator.statement
//                           ^ - invalid

